TYPE ST_Empty :
STRUCT
END_STRUCT
END_TYPE

(* stored: Version 1.1.0.1, ProductVersion 3.1.4024.15
   DUT ST_Empty: Id {51e3c0f7-65ce-4a39-9a1c-7307339c2a71} *)
